Staubli VAL3: addTraj.pgx

public program addTraj(Trajectory& x_tTrajectory)
  local num l_nSize
begin
  // mutex it
  setMutex(bActionMutex)
  if saveData:bDebug
    ? "TRAJ: Add "+x_tTrajectory.sID
  endIf
  //
  // insert a new action
  //
  if tTrajCycle.sID!="null" and tTrajCycle.sID!=""
    append(tTrajCycle)
  endIf
  // set the size
  l_nSize=size(tTrajCycle)-1
  // copy it
  tTrajCycle[l_nSize]=x_tTrajectory
  tTrajCycle[l_nSize].nId=nLastIdPoint
  // release
  bActionMutex=false
end
